TYPE ST_LaudaReadCommands_Cooling :
STRUCT
	CoolingMode	: STRING := 'IN_SP_02';
END_STRUCT
END_TYPE

(* stored: Version 1.1.0.1, ProductVersion 3.1.4024.13
   DUT ST_LaudaReadCommands_Cooling: Id {4c689db5-4aa6-45c0-b9a6-dfa7e9a6c750} *)
